TYPE ST_BaseHMIComponent_Command :
STRUCT
END_STRUCT
END_TYPE

(* stored: Version 1.1.0.1
   DUT ST_BaseHMIComponent_Command: Id {5a14d5f6-299c-05fb-0df5-3ee19b51c020} *)
